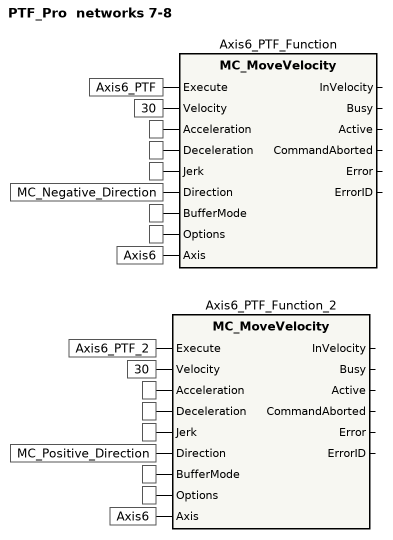
[picture p48: PTF_Pro (FBD) networks 7-8]
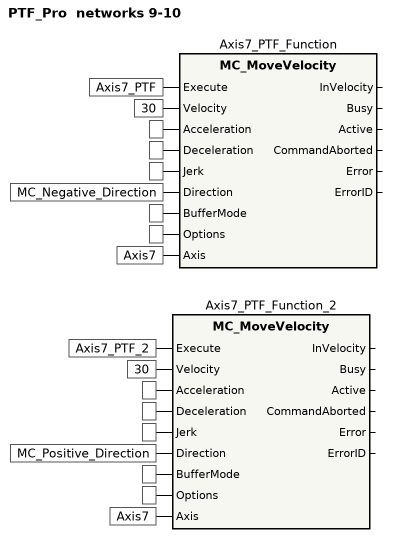
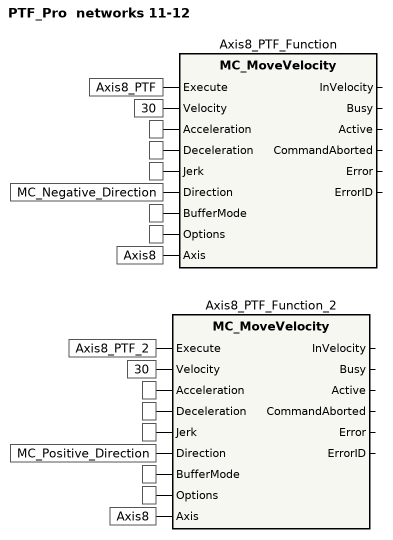
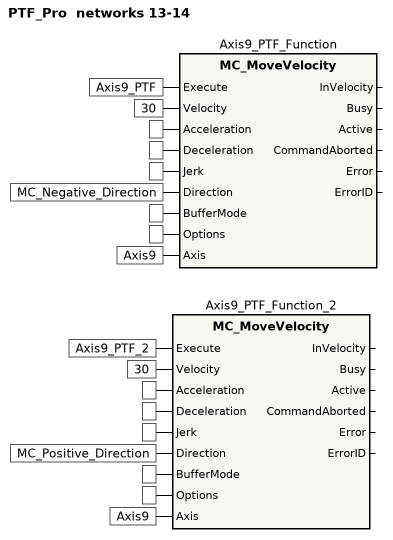
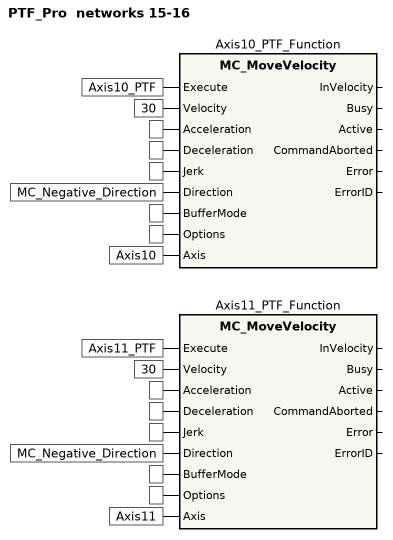
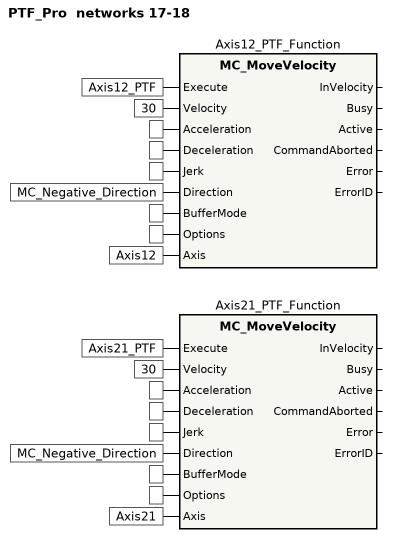
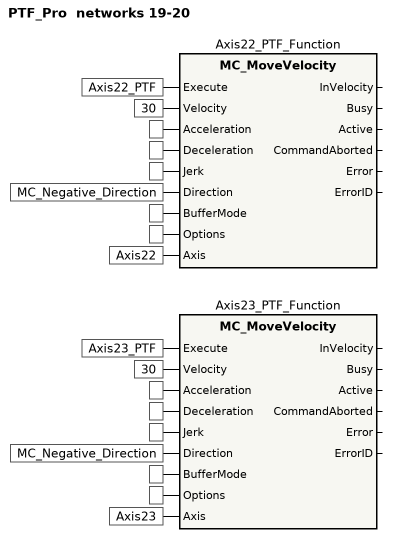
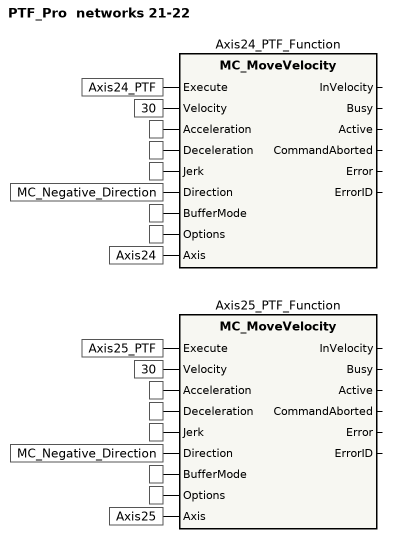
_FBD_ (* Function Block Diagram *)
NETWORK 1
	Axis1_PTF_Function:MC_MoveVelocity(Execute: Axis1_PTF, Velocity: 30, Acceleration: , Deceleration: , Jerk: , Direction: MC_Negative_Direction, BufferMode: , Options: , Axis: Axis1)
NETWORK 2
	Axis2_PTF_Function:MC_MoveVelocity(Execute: Axis2_PTF, Velocity: 30, Acceleration: , Deceleration: , Jerk: , Direction: MC_Negative_Direction, BufferMode: , Options: , Axis: Axis2)
NETWORK 3
	Axis3_PTF_Function:MC_MoveVelocity(Execute: Axis3_PTF, Velocity: 30, Acceleration: , Deceleration: , Jerk: , Direction: MC_Negative_Direction, BufferMode: , Options: , Axis: Axis3)
NETWORK 4
	Axis3_PTF_Function_2:MC_MoveVelocity(Execute: Axis3_PTF_2, Velocity: 10, Acceleration: , Deceleration: , Jerk: , Direction: MC_Positive_Direction, BufferMode: , Options: , Axis: Axis3)
NETWORK 5
	Axis4_PTF_Function:MC_MoveVelocity(Execute: Axis4_PTF, Velocity: 30, Acceleration: , Deceleration: , Jerk: , Direction: MC_Negative_Direction, BufferMode: , Options: , Axis: Axis4)
NETWORK 6
	Axis5_PTF_Function:MC_MoveVelocity(Execute: Axis5_PTF, Velocity: 30, Acceleration: , Deceleration: , Jerk: , Direction: MC_Negative_Direction, BufferMode: , Options: , Axis: Axis5)
NETWORK 7
	Axis6_PTF_Function:MC_MoveVelocity(Execute: Axis6_PTF, Velocity: 30, Acceleration: , Deceleration: , Jerk: , Direction: MC_Negative_Direction, BufferMode: , Options: , Axis: Axis6)
NETWORK 8
	Axis6_PTF_Function_2:MC_MoveVelocity(Execute: Axis6_PTF_2, Velocity: 30, Acceleration: , Deceleration: , Jerk: , Direction: MC_Positive_Direction, BufferMode: , Options: , Axis: Axis6)
NETWORK 9
	Axis7_PTF_Function:MC_MoveVelocity(Execute: Axis7_PTF, Velocity: 30, Acceleration: , Deceleration: , Jerk: , Direction: MC_Negative_Direction, BufferMode: , Options: , Axis: Axis7)
NETWORK 10
	Axis7_PTF_Function_2:MC_MoveVelocity(Execute: Axis7_PTF_2, Velocity: 30, Acceleration: , Deceleration: , Jerk: , Direction: MC_Positive_Direction, BufferMode: , Options: , Axis: Axis7)
NETWORK 11
	Axis8_PTF_Function:MC_MoveVelocity(Execute: Axis8_PTF, Velocity: 30, Acceleration: , Deceleration: , Jerk: , Direction: MC_Negative_Direction, BufferMode: , Options: , Axis: Axis8)
NETWORK 12
	Axis8_PTF_Function_2:MC_MoveVelocity(Execute: Axis8_PTF_2, Velocity: 30, Acceleration: , Deceleration: , Jerk: , Direction: MC_Positive_Direction, BufferMode: , Options: , Axis: Axis8)
NETWORK 13
	Axis9_PTF_Function:MC_MoveVelocity(Execute: Axis9_PTF, Velocity: 30, Acceleration: , Deceleration: , Jerk: , Direction: MC_Negative_Direction, BufferMode: , Options: , Axis: Axis9)
NETWORK 14
	Axis9_PTF_Function_2:MC_MoveVelocity(Execute: Axis9_PTF_2, Velocity: 30, Acceleration: , Deceleration: , Jerk: , Direction: MC_Positive_Direction, BufferMode: , Options: , Axis: Axis9)
NETWORK 15
	Axis10_PTF_Function:MC_MoveVelocity(Execute: Axis10_PTF, Velocity: 30, Acceleration: , Deceleration: , Jerk: , Direction: MC_Negative_Direction, BufferMode: , Options: , Axis: Axis10)
NETWORK 16
	Axis11_PTF_Function:MC_MoveVelocity(Execute: Axis11_PTF, Velocity: 30, Acceleration: , Deceleration: , Jerk: , Direction: MC_Negative_Direction, BufferMode: , Options: , Axis: Axis11)
NETWORK 17
	Axis12_PTF_Function:MC_MoveVelocity(Execute: Axis12_PTF, Velocity: 30, Acceleration: , Deceleration: , Jerk: , Direction: MC_Negative_Direction, BufferMode: , Options: , Axis: Axis12)
NETWORK 18
	Axis21_PTF_Function:MC_MoveVelocity(Execute: Axis21_PTF, Velocity: 30, Acceleration: , Deceleration: , Jerk: , Direction: MC_Negative_Direction, BufferMode: , Options: , Axis: Axis21)
NETWORK 19
	Axis22_PTF_Function:MC_MoveVelocity(Execute: Axis22_PTF, Velocity: 30, Acceleration: , Deceleration: , Jerk: , Direction: MC_Negative_Direction, BufferMode: , Options: , Axis: Axis22)
NETWORK 20
	Axis23_PTF_Function:MC_MoveVelocity(Execute: Axis23_PTF, Velocity: 30, Acceleration: , Deceleration: , Jerk: , Direction: MC_Negative_Direction, BufferMode: , Options: , Axis: Axis23)
NETWORK 21
	Axis24_PTF_Function:MC_MoveVelocity(Execute: Axis24_PTF, Velocity: 30, Acceleration: , Deceleration: , Jerk: , Direction: MC_Negative_Direction, BufferMode: , Options: , Axis: Axis24)
NETWORK 22
	Axis25_PTF_Function:MC_MoveVelocity(Execute: Axis25_PTF, Velocity: 30, Acceleration: , Deceleration: , Jerk: , Direction: MC_Negative_Direction, BufferMode: , Options: , Axis: Axis25)
_END_FBD_
END_PROGRAM

(* POU Other_Folder/Motion/Axis_Status_Check, FBD *)
PROGRAM Axis_Status_Check
VAR
	R1: MC_ReadStatus;
	R2: MC_ReadStatus;
	R3: MC_ReadStatus;
	R4: MC_ReadStatus;
	R5: MC_ReadStatus;
	R6: MC_ReadStatus;
	R7: MC_ReadStatus;
	R8: MC_ReadStatus;
	R9: MC_ReadStatus;
	R10: MC_ReadStatus;
	R11: MC_ReadStatus;
	R12: MC_ReadStatus;

	R21: MC_ReadStatus;
	R22: MC_ReadStatus;
	R23: MC_ReadStatus;
	R24: MC_ReadStatus;
	R25: MC_ReadStatus;
END_VAR
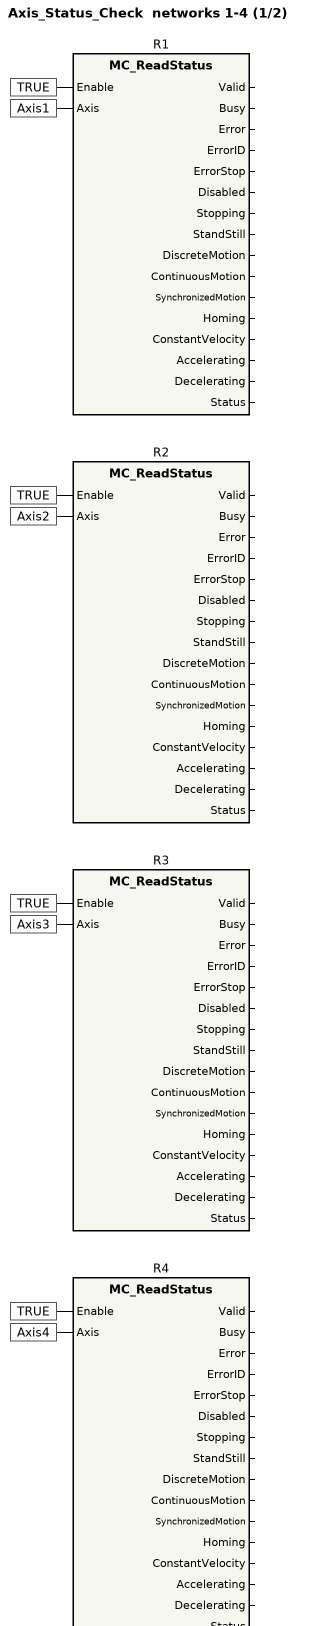
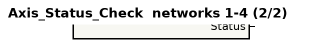
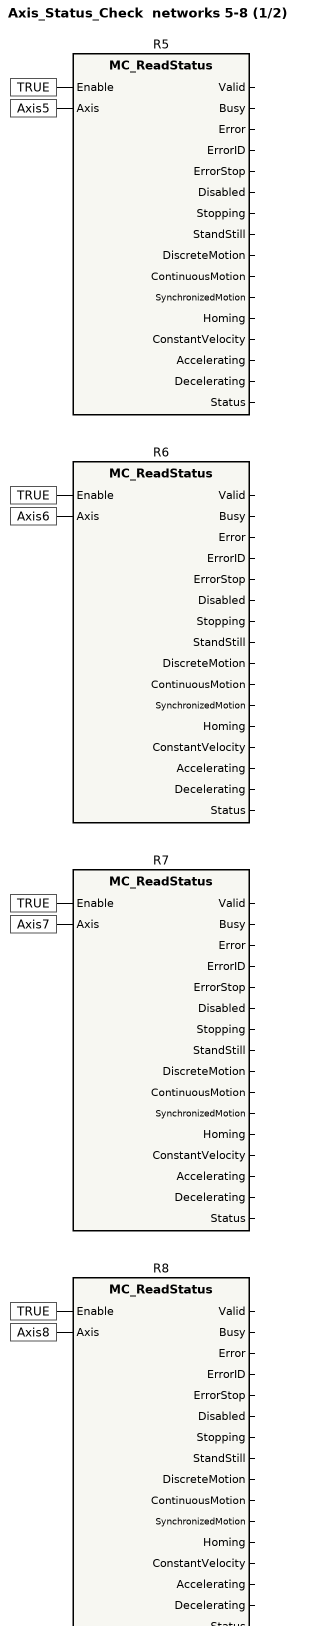
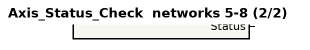
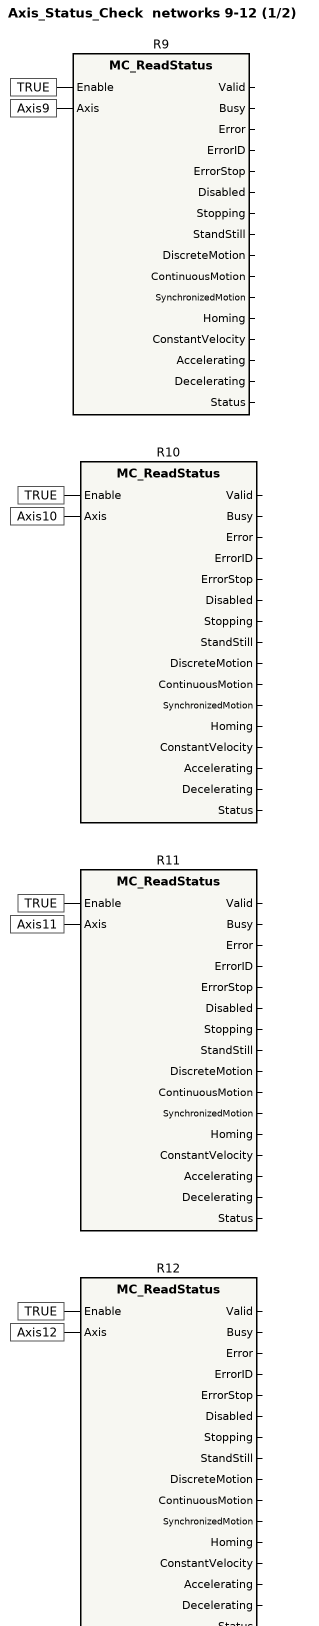
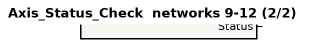
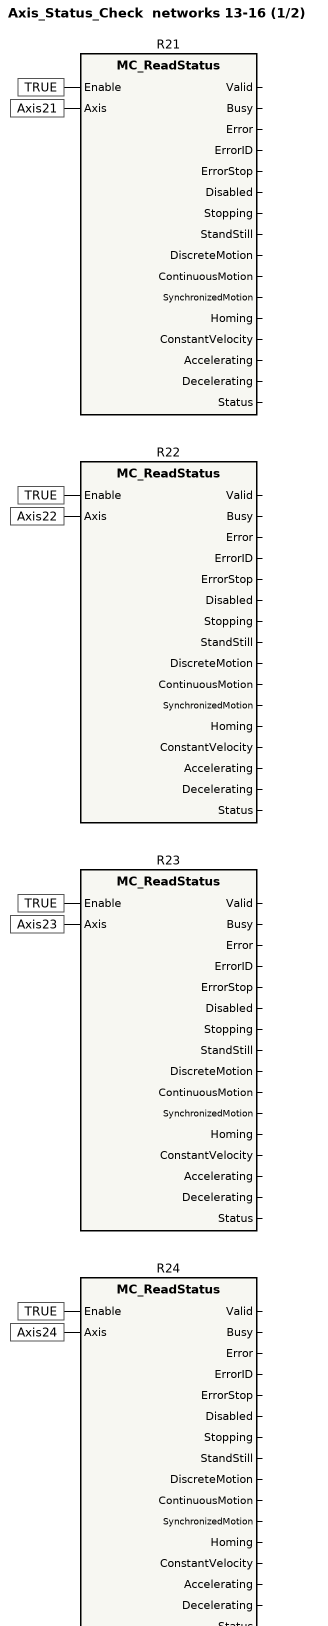
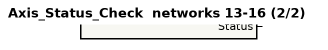
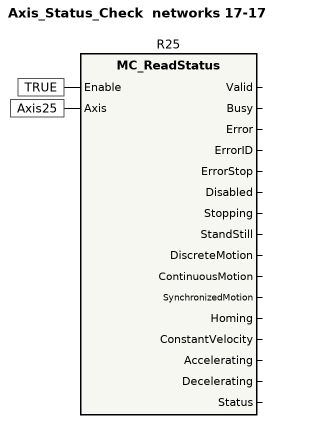
_FBD_ (* Function Block Diagram *)
NETWORK 1
	R1:MC_ReadStatus(Enable: TRUE, Axis: Axis1)
NETWORK 2
	R2:MC_ReadStatus(Enable: TRUE, Axis: Axis2)
NETWORK 3
	R3:MC_ReadStatus(Enable: TRUE, Axis: Axis3)
NETWORK 4
	R4:MC_ReadStatus(Enable: TRUE, Axis: Axis4)
NETWORK 5
	R5:MC_ReadStatus(Enable: TRUE, Axis: Axis5)
NETWORK 6
	R6:MC_ReadStatus(Enable: TRUE, Axis: Axis6)
NETWORK 7
	R7:MC_ReadStatus(Enable: TRUE, Axis: Axis7)
NETWORK 8
	R8:MC_ReadStatus(Enable: TRUE, Axis: Axis8)
NETWORK 9
	R9:MC_ReadStatus(Enable: TRUE, Axis: Axis9)
NETWORK 10
	R10:MC_ReadStatus(Enable: TRUE, Axis: Axis10)
NETWORK 11
	R11:MC_ReadStatus(Enable: TRUE, Axis: Axis11)
NETWORK 12
	R12:MC_ReadStatus(Enable: TRUE, Axis: Axis12)
NETWORK 13
	R21:MC_ReadStatus(Enable: TRUE, Axis: Axis21)
NETWORK 14
	R22:MC_ReadStatus(Enable: TRUE, Axis: Axis22)
NETWORK 15
	R23:MC_ReadStatus(Enable: TRUE, Axis: Axis23)
NETWORK 16
	R24:MC_ReadStatus(Enable: TRUE, Axis: Axis24)
NETWORK 17
	R25:MC_ReadStatus(Enable: TRUE, Axis: Axis25)
_END_FBD_
(* the same logic as Structured Text *)
(* Network 1 *)
R1(Enable := TRUE, Axis := Axis1);
(* Network 2 *)
R2(Enable := TRUE, Axis := Axis2);
(* Network 3 *)
R3(Enable := TRUE, Axis := Axis3);
(* Network 4 *)
R4(Enable := TRUE, Axis := Axis4);
(* Network 5 *)
R5(Enable := TRUE, Axis := Axis5);
(* Network 6 *)
R6(Enable := TRUE, Axis := Axis6);
(* Network 7 *)
R7(Enable := TRUE, Axis := Axis7);
(* Network 8 *)
R8(Enable := TRUE, Axis := Axis8);
(* Network 9 *)
R9(Enable := TRUE, Axis := Axis9);
(* Network 10 *)
R10(Enable := TRUE, Axis := Axis10);
(* Network 11 *)
R11(Enable := TRUE, Axis := Axis11);
(* Network 12 *)
R12(Enable := TRUE, Axis := Axis12);
(* Network 13 *)
R21(Enable := TRUE, Axis := Axis21);
(* Network 14 *)
R22(Enable := TRUE, Axis := Axis22);
(* Network 15 *)
R23(Enable := TRUE, Axis := Axis23);
(* Network 16 *)
R24(Enable := TRUE, Axis := Axis24);
(* Network 17 *)
R25(Enable := TRUE, Axis := Axis25);
END_PROGRAM

(* POU Other_Folder/Speed_AxisStatus_IO/Axis_Status, LD *)
PROGRAM Axis_Status
VAR
END_VAR
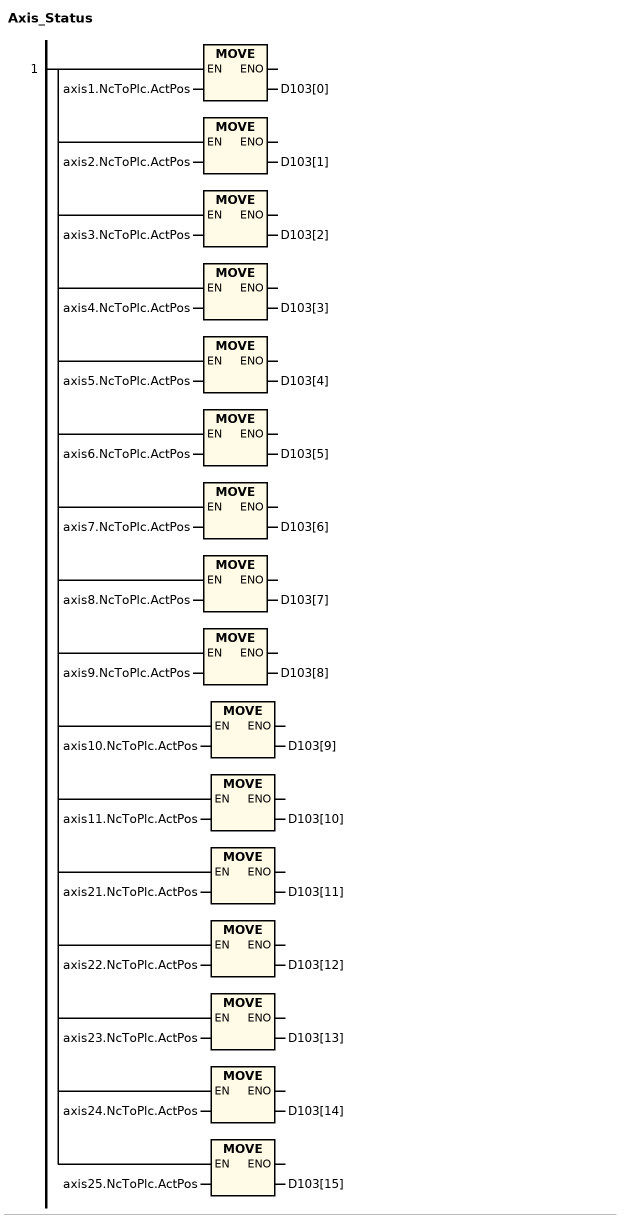
_LD_ (* Ladder Diagram *)
NETWORK 1
	*
		EN --- MOVE(axis1.NcToPlc.ActPos) => D103[0]
		EN --- MOVE(axis2.NcToPlc.ActPos) => D103[1]
		EN --- MOVE(axis3.NcToPlc.ActPos) => D103[2]
		EN --- MOVE(axis4.NcToPlc.ActPos) => D103[3]
		EN --- MOVE(axis5.NcToPlc.ActPos) => D103[4]
		EN --- MOVE(axis6.NcToPlc.ActPos) => D103[5]
		EN --- MOVE(axis7.NcToPlc.ActPos) => D103[6]
		EN --- MOVE(axis8.NcToPlc.ActPos) => D103[7]
		EN --- MOVE(axis9.NcToPlc.ActPos) => D103[8]
		EN --- MOVE(axis10.NcToPlc.ActPos) => D103[9]
		EN --- MOVE(axis11.NcToPlc.ActPos) => D103[10]
		EN --- MOVE(axis21.NcToPlc.ActPos) => D103[11]
		EN --- MOVE(axis22.NcToPlc.ActPos) => D103[12]
		EN --- MOVE(axis23.NcToPlc.ActPos) => D103[13]
		EN --- MOVE(axis24.NcToPlc.ActPos) => D103[14]
		EN --- MOVE(axis25.NcToPlc.ActPos) => D103[15]
_END_LD_
(* the same logic as Structured Text *)
(* Network 1 *)
D103[0] := axis1.NcToPlc.ActPos;
D103[1] := axis2.NcToPlc.ActPos;
D103[2] := axis3.NcToPlc.ActPos;
D103[3] := axis4.NcToPlc.ActPos;
D103[4] := axis5.NcToPlc.ActPos;
D103[5] := axis6.NcToPlc.ActPos;
D103[6] := axis7.NcToPlc.ActPos;
D103[7] := axis8.NcToPlc.ActPos;
D103[8] := axis9.NcToPlc.ActPos;
D103[9] := axis10.NcToPlc.ActPos;
D103[10] := axis11.NcToPlc.ActPos;
D103[11] := axis21.NcToPlc.ActPos;
D103[12] := axis22.NcToPlc.ActPos;
D103[13] := axis23.NcToPlc.ActPos;
D103[14] := axis24.NcToPlc.ActPos;
D103[15] := axis25.NcToPlc.ActPos;
END_PROGRAM

(* POU Other_Folder/Speed_AxisStatus_IO/Limit_Mapping, LD *)
PROGRAM Limit_Mapping
VAR

END_VAR
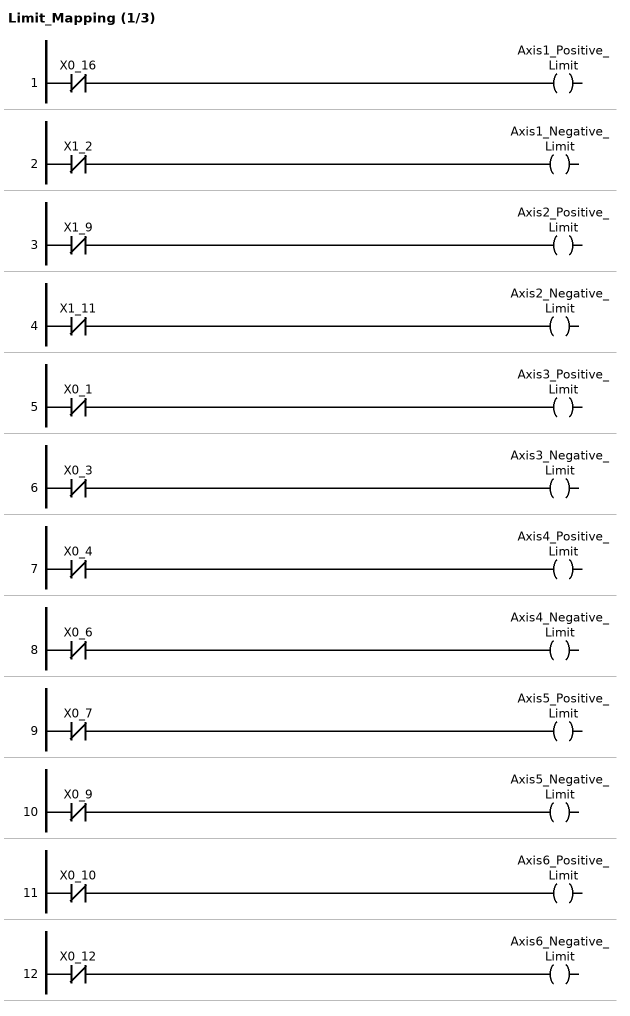
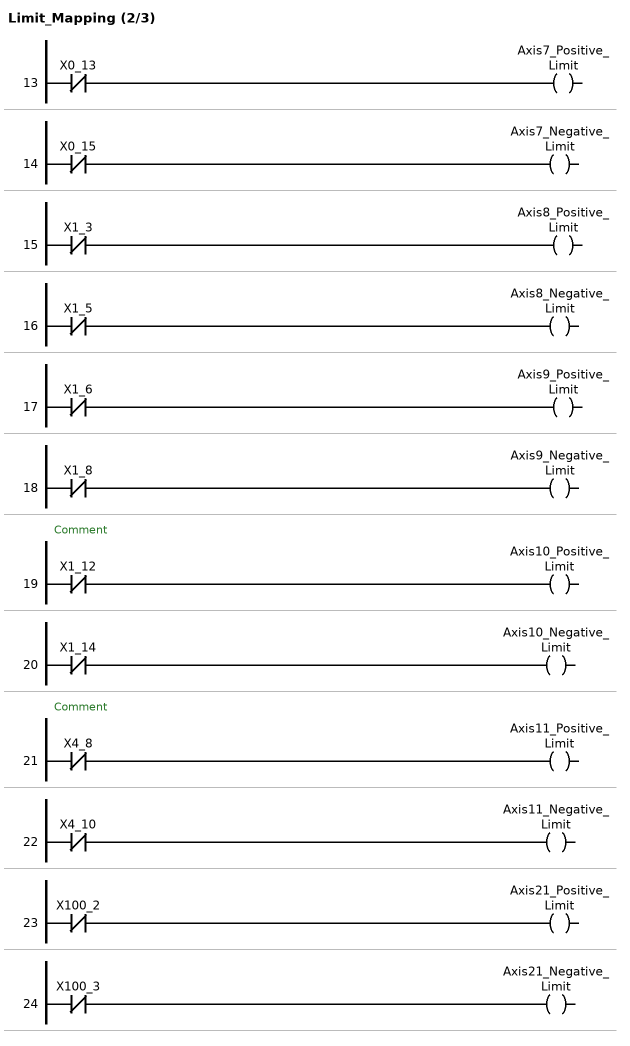
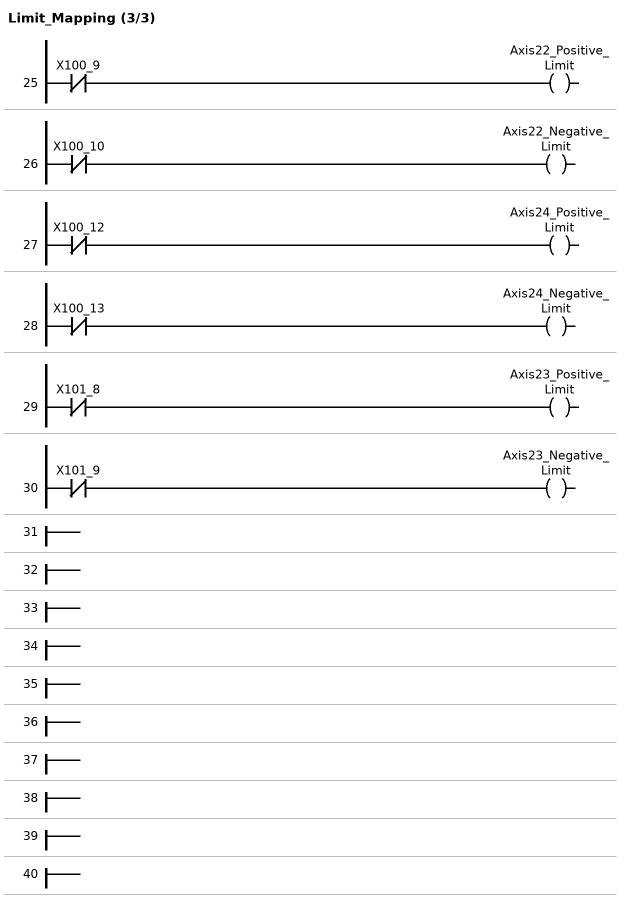
_LD_ (* Ladder Diagram *)
NETWORK 1
	[/X0_16] --- (Axis1_Positive_Limit)
NETWORK 2
	[/X1_2] --- (Axis1_Negative_Limit)
NETWORK 3
	[/X1_9] --- (Axis2_Positive_Limit)
NETWORK 4
	[/X1_11] --- (Axis2_Negative_Limit)
NETWORK 5
	[/X0_1] --- (Axis3_Positive_Limit)
NETWORK 6
	[/X0_3] --- (Axis3_Negative_Limit)
NETWORK 7
	[/X0_4] --- (Axis4_Positive_Limit)
NETWORK 8
	[/X0_6] --- (Axis4_Negative_Limit)
NETWORK 9
	[/X0_7] --- (Axis5_Positive_Limit)
NETWORK 10
	[/X0_9] --- (Axis5_Negative_Limit)
NETWORK 11
	[/X0_10] --- (Axis6_Positive_Limit)
NETWORK 12
	[/X0_12] --- (Axis6_Negative_Limit)
NETWORK 13
	[/X0_13] --- (Axis7_Positive_Limit)
NETWORK 14
	[/X0_15] --- (Axis7_Negative_Limit)
NETWORK 15
	[/X1_3] --- (Axis8_Positive_Limit)
NETWORK 16
	[/X1_5] --- (Axis8_Negative_Limit)
NETWORK 17
	[/X1_6] --- (Axis9_Positive_Limit)
NETWORK 18
	[/X1_8] --- (Axis9_Negative_Limit)
NETWORK 19 (* Comment *)
	[/X1_12] --- (Axis10_Positive_Limit)
NETWORK 20
	[/X1_14] --- (Axis10_Negative_Limit)
NETWORK 21 (* Comment *)
	[/X4_8] --- (Axis11_Positive_Limit)
NETWORK 22
	[/X4_10] --- (Axis11_Negative_Limit)
NETWORK 23
	[/X100_2] --- (Axis21_Positive_Limit)
NETWORK 24
	[/X100_3] --- (Axis21_Negative_Limit)
NETWORK 25
	[/X100_9] --- (Axis22_Positive_Limit)
NETWORK 26
	[/X100_10] --- (Axis22_Negative_Limit)
NETWORK 27
	[/X100_12] --- (Axis24_Positive_Limit)
NETWORK 28
	[/X100_13] --- (Axis24_Negative_Limit)
NETWORK 29
	[/X101_8] --- (Axis23_Positive_Limit)
NETWORK 30
	[/X101_9] --- (Axis23_Negative_Limit)
NETWORK 31
	*
NETWORK 32
	*
NETWORK 33
	*
NETWORK 34
	*
NETWORK 35
	*
NETWORK 36
	*
NETWORK 37
	*
NETWORK 38
	*
NETWORK 39
	*
NETWORK 40
	*
_END_LD_
(* the same logic as Structured Text *)
(* Network 1 *)
Axis1_Positive_Limit := NOT X0_16;
(* Network 2 *)
Axis1_Negative_Limit := NOT X1_2;
(* Network 3 *)
Axis2_Positive_Limit := NOT X1_9;
(* Network 4 *)
Axis2_Negative_Limit := NOT X1_11;
(* Network 5 *)
Axis3_Positive_Limit := NOT X0_1;
(* Network 6 *)
Axis3_Negative_Limit := NOT X0_3;
(* Network 7 *)
Axis4_Positive_Limit := NOT X0_4;
(* Network 8 *)
Axis4_Negative_Limit := NOT X0_6;
(* Network 9 *)
Axis5_Positive_Limit := NOT X0_7;
(* Network 10 *)
Axis5_Negative_Limit := NOT X0_9;
(* Network 11 *)
Axis6_Positive_Limit := NOT X0_10;
(* Network 12 *)
Axis6_Negative_Limit := NOT X0_12;
(* Network 13 *)
Axis7_Positive_Limit := NOT X0_13;
(* Network 14 *)
Axis7_Negative_Limit := NOT X0_15;
(* Network 15 *)
Axis8_Positive_Limit := NOT X1_3;
(* Network 16 *)
Axis8_Negative_Limit := NOT X1_5;
(* Network 17 *)
Axis9_Positive_Limit := NOT X1_6;
(* Network 18 *)
Axis9_Negative_Limit := NOT X1_8;
(* Network 19: Comment *)
Axis10_Positive_Limit := NOT X1_12;
(* Network 20 *)
Axis10_Negative_Limit := NOT X1_14;
(* Network 21: Comment *)
Axis11_Positive_Limit := NOT X4_8;
(* Network 22 *)
Axis11_Negative_Limit := NOT X4_10;
(* Network 23 *)
Axis21_Positive_Limit := NOT X100_2;
(* Network 24 *)
Axis21_Negative_Limit := NOT X100_3;
(* Network 25 *)
Axis22_Positive_Limit := NOT X100_9;
(* Network 26 *)
Axis22_Negative_Limit := NOT X100_10;
(* Network 27 *)
Axis24_Positive_Limit := NOT X100_12;
(* Network 28 *)
Axis24_Negative_Limit := NOT X100_13;
(* Network 29 *)
Axis23_Positive_Limit := NOT X101_8;
(* Network 30 *)
Axis23_Negative_Limit := NOT X101_9;
(* Network 31 *)
(* Network 32 *)
(* Network 33 *)
(* Network 34 *)
(* Network 35 *)
(* Network 36 *)
(* Network 37 *)
(* Network 38 *)
(* Network 39 *)
(* Network 40 *)
END_PROGRAM

(* POU Other_Folder/Speed_AxisStatus_IO/Speed_Setting, ST *)
PROGRAM Speed_Setting
VAR
	UP1: R_TRIG;
	UP2: R_TRIG;
	UP3: R_TRIG;

	step: INT;
END_VAR
CASE step OF
0:
step:=1;

1:
UP1(CLK:=M100 , Q=> );
UP2(CLK:=M101 , Q=> );
UP3(CLK:=M102 , Q=> );
(*调速选择*)
IF UP1.Q THEN(*低速*)
D11:=D100[0];D12:=D100[1];D13:=D100[2];D14:=D100[3];D15:=D100[4];
D16:=D100[5];D17:=D100[6];D18:=D100[7];D19:=D100[8];D20:=D100[9];D2_1:=D100[10];
V211:=D100[11];V221:=D100[12];V231:=D100[13];V241:=D100[14];V251:=D100[15];
step:=10;
END_IF
IF UP2.Q THEN(*中速*)
D11:=D101[0];D12:=D101[1];D13:=D101[2];D14:=D101[3];D15:=D101[4];
D16:=D101[5];D17:=D101[6];D18:=D101[7];D19:=D101[8];D20:=D101[9];D2_1:=D101[10];
V211:=D101[11];V221:=D101[12];V231:=D101[13];V241:=D101[14];V251:=D101[15];
step:=20;
END_IF
IF UP3.Q THEN(*高速*)
D11:=D102[0];D12:=D102[1];D13:=D102[2];D14:=D102[3];D15:=D102[4];
D16:=D102[5];D17:=D102[6];D18:=D102[7];D19:=D102[8];D20:=D102[9];D2_1:=D102[10];
V211:=D102[11];V221:=D102[12];V231:=D102[13];V241:=D102[14];V251:=D102[15];
step:=30;
END_IF

10:
M101:=FALSE;
M102:=FALSE;
step:=1;

20:
M100:=FALSE;
M102:=FALSE;
step:=1;

30:
M100:=FALSE;
M101:=FALSE;
step:=1;

END_CASE
END_PROGRAM

(* POU Debug_Folder/Axis1_Debug_Model, ST *)
PROGRAM Axis1_Debug_Model
VAR
	UP1: R_TRIG;
	UP2: R_TRIG;
	UP3: R_TRIG;
	UP4: R_TRIG;
	step:INT;
END_VAR
UP1(CLK:=Axis1_debug_trigger , Q=> );

CASE step OF
0:
IF UP1.Q THEN
step:=1;
END_IF;

1:
(*点动加-----------
点动减------------
手动点动-----------*)
UP2(CLK:=Axis1_mov_add , Q=> );
UP3(CLK:=Axis1_mov_sub , Q=> );
UP4(CLK:=Axis1_mov_line , Q=> );

IF UP2.Q AND Debug_Model AND Axis1_Poweron AND NOT Total_Pause THEN
D1:=Axis1.NcToPlc.ActPos+D200;
Axis1_mov_add:=FALSE;
step:=10;
ELSE
Axis1_mov_add:=FALSE;
Axis1_MoveAbsolute:=FALSE;
END_IF

IF UP3.Q AND Debug_Model AND Axis1_Poweron AND NOT Total_Pause THEN
D1:=Axis1.NcToPlc.ActPos-D200;
Axis1_mov_sub:=FALSE;
step:=10;
ELSE
Axis1_mov_sub:=FALSE;
Axis1_MoveAbsolute:=FALSE;
END_IF

IF UP4.Q AND Debug_Model AND Axis1_Poweron  AND NOT Total_Pause THEN
D1:=D201;
Axis1_mov_line:=FALSE;
step:=10;
ELSE
Axis1_mov_line:=FALSE;
Axis1_MoveAbsolute:=FALSE;
END_IF

10:
Axis1_MoveAbsolute:=TRUE;
IF Axis1_Abs_Function.Done THEN
Axis1_MoveAbsolute:=FALSE;
step:=1;
END_IF

END_CASE

IF Axis1_mov_add THEN
Axis1_mov_add:=FALSE;
END_IF
IF Axis1_mov_sub THEN
Axis1_mov_sub:=FALSE;
END_IF
IF Axis1_mov_line THEN
Axis1_mov_line:=FALSE;
END_IF


IF NOT Debug_Model  THEN
Axis1_debug_trigger:=FALSE;
step:=0;
END_IF

IF Total_Emergency THEN
Axis1_debug_trigger:=FALSE;
Axis1_mov_add:=FALSE;
Axis1_mov_sub:=FALSE;
Axis1_mov_line:=FALSE;
Axis1_MoveAbsolute:=FALSE;
step:=0;
END_IF
END_PROGRAM

(* POU Debug_Folder/Axis2_Debug_Model, ST *)
PROGRAM Axis2_Debug_Model
VAR
	UP1: R_TRIG;
	UP2: R_TRIG;
	UP3: R_TRIG;
	UP4: R_TRIG;
	step:INT;

END_VAR
UP1(CLK:=Axis2_debug_trigger , Q=> );

CASE step OF
0:
IF UP1.Q THEN
step:=1;
END_IF;

1:
UP2(CLK:=Axis2_mov_add , Q=> );
UP3(CLK:=Axis2_mov_sub , Q=> );
UP4(CLK:=Axis2_mov_line , Q=> );

IF UP2.Q AND Debug_Model AND Axis2_Poweron AND NOT Total_Pause THEN
D2:=Axis2.NcToPlc.ActPos+D200;
Axis2_mov_add:=FALSE;
step:=10;
ELSE
Axis2_mov_add:=FALSE;
Axis2_MoveAbsolute:=FALSE;
END_IF

IF UP3.Q AND Debug_Model AND Axis2_Poweron AND NOT Total_Pause THEN
D2:=Axis2.NcToPlc.ActPos-D200;
Axis2_mov_sub:=FALSE;
step:=10;
ELSE
Axis2_mov_sub:=FALSE;
Axis2_MoveAbsolute:=FALSE;
END_IF

IF UP4.Q AND Debug_Model AND Axis2_Poweron AND NOT Total_Pause THEN
D2:=D202;
Axis2_mov_line:=FALSE;
step:=10;
ELSE
Axis2_mov_line:=FALSE;
Axis2_MoveAbsolute:=FALSE;
END_IF

10:
Axis2_MoveAbsolute:=TRUE;
IF Axis2_Abs_Function.Done THEN
Axis2_MoveAbsolute:=FALSE;
step:=1;
END_IF

END_CASE

IF Axis2_mov_add THEN
Axis2_mov_add:=FALSE;
END_IF
IF Axis2_mov_sub THEN
Axis2_mov_sub:=FALSE;
END_IF
IF Axis2_mov_line THEN
Axis2_mov_line:=FALSE;
END_IF


IF NOT Debug_Model  THEN
Axis2_debug_trigger:=FALSE;
step:=0;
END_IF

IF Total_Emergency THEN
Axis2_debug_trigger:=FALSE;
Axis2_mov_add:=FALSE;
Axis2_mov_sub:=FALSE;
Axis2_mov_line:=FALSE;
Axis2_MoveAbsolute:=FALSE;
step:=0;
END_IF
END_PROGRAM

(* POU Debug_Folder/Axis3_Debug_Model, ST *)
PROGRAM Axis3_Debug_Model
VAR
	UP1: R_TRIG;
	UP2: R_TRIG;
	UP3: R_TRIG;
	UP4: R_TRIG;
	step:INT;
END_VAR
UP1(CLK:=Axis3_debug_trigger , Q=> );

CASE step OF
0:
IF UP1.Q THEN
step:=1;
END_IF;

1:
UP2(CLK:=Axis3_mov_add , Q=> );
UP3(CLK:=Axis3_mov_sub , Q=> );
UP4(CLK:=Axis3_mov_line , Q=> );

IF UP2.Q AND Debug_Model AND Axis3_Poweron AND NOT Total_Pause THEN
D3:=Axis3.NcToPlc.ActPos+D200;
Axis3_mov_add:=FALSE;
step:=10;
ELSE
Axis3_mov_add:=FALSE;
Axis3_MoveAbsolute:=FALSE;
END_IF

IF UP3.Q AND Debug_Model AND Axis3_Poweron AND NOT Total_Pause THEN
D3:=Axis3.NcToPlc.ActPos-D200;
Axis3_mov_sub:=FALSE;
step:=10;
ELSE
Axis3_mov_sub:=FALSE;
Axis3_MoveAbsolute:=FALSE;
END_IF

IF UP4.Q AND Debug_Model AND Axis3_Poweron AND NOT Total_Pause THEN
D3:=D203;
Axis3_mov_line:=FALSE;
step:=10;
ELSE
Axis3_mov_line:=FALSE;
Axis3_MoveAbsolute:=FALSE;
END_IF

10:
Axis3_MoveAbsolute:=TRUE;
IF Axis3_Abs_Function.Done THEN
Axis3_MoveAbsolute:=FALSE;
step:=1;
END_IF

END_CASE

IF Axis3_mov_add THEN
Axis3_mov_add:=FALSE;
END_IF
IF Axis3_mov_sub THEN
Axis3_mov_sub:=FALSE;
END_IF
IF Axis3_mov_line THEN
Axis3_mov_line:=FALSE;
END_IF


IF NOT Debug_Model  THEN
Axis3_debug_trigger:=FALSE;
step:=0;
END_IF

IF Total_Emergency THEN
Axis3_debug_trigger:=FALSE;
Axis3_mov_add:=FALSE;
Axis3_mov_sub:=FALSE;
Axis3_mov_line:=FALSE;
Axis3_MoveAbsolute:=FALSE;
step:=0;
END_IF
END_PROGRAM

(* POU Debug_Folder/Axis4_Debug_Model, ST *)
PROGRAM Axis4_Debug_Model
VAR
	UP1: R_TRIG;
	UP2: R_TRIG;
	UP3: R_TRIG;
	UP4: R_TRIG;
	step:INT;
	M1:BOOL;


END_VAR
UP1(CLK:=Axis4_debug_trigger , Q=> );

CASE step OF
0:
IF UP1.Q THEN
step:=1;
END_IF;

1:
UP2(CLK:=Axis4_mov_add , Q=> );
IF UP2.Q AND Debug_Model AND Axis4_Poweron  AND NOT Total_Pause THEN
D4:=Axis4.NcToPlc.ActPos+D200;
Axis4_mov_add:=FALSE;
step:=10;
ELSE
Axis4_mov_add:=FALSE;
Axis4_MoveAbsolute:=FALSE;
END_IF


UP3(CLK:=Axis4_mov_sub , Q=> );
IF UP3.Q AND Debug_Model AND Axis4_Poweron  AND NOT Total_Pause  THEN
D4:=Axis4.NcToPlc.ActPos-D200;
Axis4_mov_sub:=FALSE;
step:=10;
ELSE
Axis4_mov_sub:=FALSE;
Axis4_MoveAbsolute:=FALSE;
END_IF


UP4(CLK:=Axis4_mov_line , Q=> );
IF UP4.Q AND Debug_Model AND Axis4_Poweron  AND NOT Total_Pause  THEN
D4:=D204;
Axis4_mov_line:=FALSE;
step:=10;
ELSE
Axis4_mov_line:=FALSE;
Axis4_MoveAbsolute:=FALSE;
END_IF


10:
Axis4_MoveAbsolute:=TRUE;
IF Axis4_Abs_Function.Done THEN
Axis4_MoveAbsolute:=FALSE;
step:=1;
END_IF


END_CASE

IF Axis4_mov_add THEN
Axis4_mov_add:=FALSE;
END_IF
IF Axis4_mov_sub THEN
Axis4_mov_sub:=FALSE;
END_IF
IF Axis4_mov_line THEN
Axis4_mov_line:=FALSE;
END_IF


IF NOT Debug_Model  THEN
Axis4_debug_trigger:=FALSE;
step:=0;
END_IF

IF Total_Emergency THEN
Axis4_debug_trigger:=FALSE;
Axis4_mov_add:=FALSE;
Axis4_mov_sub:=FALSE;
Axis4_mov_line:=FALSE;
Axis4_MoveAbsolute:=FALSE;
Axis4_1_MoveAbsolute:=FALSE;
step:=0;
END_IF
END_PROGRAM

(* POU Debug_Folder/Axis5_Debug_Model, ST *)
PROGRAM Axis5_Debug_Model
VAR
	UP1: R_TRIG;
	UP2: R_TRIG;
	UP3: R_TRIG;
	UP4: R_TRIG;
	step:INT;
END_VAR
UP1(CLK:=Axis5_debug_trigger , Q=> );

CASE step OF
0:
IF UP1.Q THEN
step:=1;
END_IF;

1:
UP2(CLK:=Axis5_mov_add , Q=> );
UP3(CLK:=Axis5_mov_sub , Q=> );
UP4(CLK:=Axis5_mov_line , Q=> );

IF UP2.Q AND Debug_Model AND Axis5_Poweron  AND NOT Total_Pause THEN
D5:=Axis5.NcToPlc.ActPos+D200;
Axis5_mov_add:=FALSE;
step:=10;
ELSE
Axis5_mov_add:=FALSE;
Axis5_MoveAbsolute:=FALSE;
END_IF

IF UP3.Q AND Debug_Model AND Axis5_Poweron AND NOT Total_Pause THEN
D5:=Axis5.NcToPlc.ActPos-D200;
Axis5_mov_sub:=FALSE;
step:=10;
ELSE
Axis5_mov_sub:=FALSE;
Axis5_MoveAbsolute:=FALSE;
END_IF

IF UP4.Q AND Debug_Model AND Axis5_Poweron  AND NOT Total_Pause THEN
D5:=D205;
Axis5_mov_line:=FALSE;
step:=10;
ELSE
Axis5_mov_line:=FALSE;
Axis5_MoveAbsolute:=FALSE;
END_IF

10:
Axis5_MoveAbsolute:=TRUE;
IF Axis5_Abs_Function.Done THEN
Axis5_MoveAbsolute:=FALSE;
step:=1;
END_IF

END_CASE

IF Axis5_mov_add THEN
Axis5_mov_add:=FALSE;
END_IF
IF Axis5_mov_sub THEN
Axis5_mov_sub:=FALSE;
END_IF
IF Axis5_mov_line THEN
Axis5_mov_line:=FALSE;
END_IF


IF NOT Debug_Model  THEN
Axis5_debug_trigger:=FALSE;
step:=0;
END_IF

IF Total_Emergency THEN
Axis5_debug_trigger:=FALSE;
Axis5_mov_add:=FALSE;
Axis5_mov_sub:=FALSE;
Axis5_mov_line:=FALSE;
Axis5_MoveAbsolute:=FALSE;
Axis5_1_MoveAbsolute:=FALSE;
step:=0;
END_IF
END_PROGRAM

(* POU Debug_Folder/Axis6_Debug_Model, ST *)
PROGRAM Axis6_Debug_Model
VAR
	UP1: R_TRIG;
	UP2: R_TRIG;
	UP3: R_TRIG;
	UP4: R_TRIG;
	step:INT;
END_VAR
UP1(CLK:=Axis6_debug_trigger , Q=> );

CASE step OF
0:
IF UP1.Q THEN
step:=1;
END_IF;

1:
UP2(CLK:=Axis6_mov_add , Q=> );
UP3(CLK:=Axis6_mov_sub , Q=> );
UP4(CLK:=Axis6_mov_line , Q=> );

IF UP2.Q AND Debug_Model AND Axis6_Poweron  AND NOT Total_Pause THEN
D6:=Axis6.NcToPlc.ActPos+D200;
Axis6_mov_add:=FALSE;
step:=10;
ELSE
Axis6_mov_add:=FALSE;
Axis6_MoveAbsolute:=FALSE;
END_IF

IF UP3.Q AND Debug_Model AND Axis6_Poweron AND NOT Total_Pause THEN
D6:=Axis6.NcToPlc.ActPos-D200;
Axis6_mov_sub:=FALSE;
step:=10;
ELSE
Axis6_mov_sub:=FALSE;
Axis6_MoveAbsolute:=FALSE;
END_IF

IF UP4.Q AND Debug_Model AND Axis6_Poweron  AND NOT Total_Pause THEN
D6:=D206;
Axis6_mov_line:=FALSE;
step:=10;
ELSE
Axis6_mov_line:=FALSE;
Axis6_MoveAbsolute:=FALSE;
END_IF

10:
Axis6_MoveAbsolute:=TRUE;
IF Axis6_Abs_Function.Done THEN
Axis6_MoveAbsolute:=FALSE;
step:=1;
END_IF
END_CASE

IF Axis6_mov_add THEN
Axis6_mov_add:=FALSE;
END_IF
IF Axis6_mov_sub THEN
Axis6_mov_sub:=FALSE;
END_IF
IF Axis6_mov_line THEN
Axis6_mov_line:=FALSE;
END_IF


IF NOT Debug_Model  THEN
Axis6_debug_trigger:=FALSE;
step:=0;
END_IF

IF Total_Emergency THEN
Axis6_debug_trigger:=FALSE;
Axis6_mov_add:=FALSE;
Axis6_mov_sub:=FALSE;
Axis6_mov_line:=FALSE;
Axis6_MoveAbsolute:=FALSE;
step:=0;
END_IF
END_PROGRAM

(* POU Debug_Folder/Axis7_Debug_Model, ST *)
PROGRAM Axis7_Debug_Model
VAR
	UP1: R_TRIG;
	UP2: R_TRIG;
	UP3: R_TRIG;
	UP4: R_TRIG;
	step:INT;
END_VAR
UP1(CLK:=Axis7_debug_trigger , Q=> );

CASE step OF
0:
IF UP1.Q THEN
step:=1;
END_IF;

1:
UP2(CLK:=Axis7_mov_add , Q=> );
UP3(CLK:=Axis7_mov_sub , Q=> );
UP4(CLK:=Axis7_mov_line , Q=> );

IF UP2.Q AND Debug_Model AND Axis7_Poweron  AND NOT Total_Pause THEN
D7:=Axis7.NcToPlc.ActPos+D200;
Axis7_mov_add:=FALSE;
step:=10;
ELSE
Axis7_mov_add:=FALSE;
Axis7_MoveAbsolute:=FALSE;
END_IF

IF UP3.Q AND Debug_Model AND Axis7_Poweron AND NOT Total_Pause THEN
D7:=Axis7.NcToPlc.ActPos-D200;
Axis7_mov_sub:=FALSE;
step:=10;
ELSE
Axis7_mov_sub:=FALSE;
Axis7_MoveAbsolute:=FALSE;
END_IF

IF UP4.Q AND Debug_Model AND Axis7_Poweron  AND NOT Total_Pause THEN
D7:=D207;
Axis7_mov_line:=FALSE;
step:=10;
ELSE
Axis7_mov_line:=FALSE;
Axis7_MoveAbsolute:=FALSE;
END_IF

10:
Axis7_MoveAbsolute:=TRUE;
IF Axis7_Abs_Function.Done THEN
Axis7_MoveAbsolute:=FALSE;
step:=1;
END_IF
END_CASE

IF Axis7_mov_add THEN
Axis7_mov_add:=FALSE;
END_IF
IF Axis7_mov_sub THEN
Axis7_mov_sub:=FALSE;
END_IF
IF Axis7_mov_line THEN
Axis7_mov_line:=FALSE;
END_IF


IF NOT Debug_Model  THEN
Axis7_debug_trigger:=FALSE;
step:=0;
END_IF

IF Total_Emergency THEN
Axis7_debug_trigger:=FALSE;
Axis7_mov_add:=FALSE;
Axis7_mov_sub:=FALSE;
Axis7_mov_line:=FALSE;
Axis7_MoveAbsolute:=FALSE;
step:=0;
END_IF
END_PROGRAM

(* POU Debug_Folder/Axis8_Debug_Model, ST *)
PROGRAM Axis8_Debug_Model
VAR
	UP1: R_TRIG;
	UP2: R_TRIG;
	UP3: R_TRIG;
	UP4: R_TRIG;
	step:INT;
END_VAR
UP1(CLK:=Axis8_debug_trigger , Q=> );

CASE step OF
0:
IF UP1.Q THEN
step:=1;
END_IF;

1:
UP2(CLK:=Axis8_mov_add , Q=> );
UP3(CLK:=Axis8_mov_sub , Q=> );
UP4(CLK:=Axis8_mov_line , Q=> );

IF UP2.Q AND Debug_Model AND Axis8_Poweron  AND NOT Total_Pause THEN
D8:=Axis8.NcToPlc.ActPos+D200;
Axis8_mov_add:=FALSE;
step:=10;
ELSE
Axis8_mov_add:=FALSE;
Axis8_MoveAbsolute:=FALSE;
END_IF

IF UP3.Q AND Debug_Model AND Axis8_Poweron AND NOT Total_Pause THEN
D8:=Axis8.NcToPlc.ActPos-D200;
Axis8_mov_sub:=FALSE;
step:=10;
ELSE
Axis8_mov_sub:=FALSE;
Axis8_MoveAbsolute:=FALSE;
END_IF

IF UP4.Q AND Debug_Model AND Axis8_Poweron  AND NOT Total_Pause THEN
D8:=D208;
Axis8_mov_line:=FALSE;
step:=10;
ELSE
Axis8_mov_line:=FALSE;
Axis8_MoveAbsolute:=FALSE;
END_IF

10:
Axis8_MoveAbsolute:=TRUE;
IF Axis8_Abs_Function.Done THEN
Axis8_MoveAbsolute:=FALSE;
step:=1;
END_IF
END_CASE

IF Axis8_mov_add THEN
Axis8_mov_add:=FALSE;
END_IF
IF Axis8_mov_sub THEN
Axis8_mov_sub:=FALSE;
END_IF
IF Axis8_mov_line THEN
Axis8_mov_line:=FALSE;
END_IF


IF NOT Debug_Model  THEN
Axis8_debug_trigger:=FALSE;
step:=0;
END_IF

IF Total_Emergency THEN
Axis8_debug_trigger:=FALSE;
Axis8_mov_add:=FALSE;
Axis8_mov_sub:=FALSE;
Axis8_mov_line:=FALSE;
Axis8_MoveAbsolute:=FALSE;
step:=0;
END_IF
END_PROGRAM

(* POU Debug_Folder/Axis9_Debug_Model, ST *)
PROGRAM Axis9_Debug_Model
VAR
	UP1: R_TRIG;
	UP2: R_TRIG;
	UP3: R_TRIG;
	UP4: R_TRIG;
	step:INT;
END_VAR
UP1(CLK:=Axis9_debug_trigger , Q=> );

CASE step OF
0:
IF UP1.Q THEN
step:=1;
END_IF;

1:
UP2(CLK:=Axis9_mov_add , Q=> );
UP3(CLK:=Axis9_mov_sub , Q=> );
UP4(CLK:=Axis9_mov_line , Q=> );

IF UP2.Q AND Debug_Model AND Axis9_Poweron  AND NOT Total_Pause THEN
D9:=Axis9.NcToPlc.ActPos+D200;
Axis9_mov_add:=FALSE;
step:=10;
ELSE
Axis9_mov_add:=FALSE;
Axis9_MoveAbsolute:=FALSE;
END_IF

IF UP3.Q AND Debug_Model AND Axis9_Poweron AND NOT Total_Pause THEN
D9:=Axis9.NcToPlc.ActPos-D200;
Axis9_mov_sub:=FALSE;
step:=10;
ELSE
Axis9_mov_sub:=FALSE;
Axis9_MoveAbsolute:=FALSE;
END_IF

IF UP4.Q AND Debug_Model AND Axis9_Poweron  AND NOT Total_Pause THEN
D9:=D209;
Axis9_mov_line:=FALSE;
step:=10;
ELSE
Axis9_mov_line:=FALSE;
Axis9_MoveAbsolute:=FALSE;
END_IF

10:
Axis9_MoveAbsolute:=TRUE;
IF Axis9_Abs_Function.Done THEN
Axis9_MoveAbsolute:=FALSE;
step:=1;
END_IF
END_CASE

IF Axis9_mov_add THEN
Axis9_mov_add:=FALSE;
END_IF
IF Axis9_mov_sub THEN
Axis9_mov_sub:=FALSE;
END_IF
IF Axis9_mov_line THEN
Axis9_mov_line:=FALSE;
END_IF


IF NOT Debug_Model  THEN
Axis9_debug_trigger:=FALSE;
step:=0;
END_IF

IF Total_Emergency THEN
Axis9_debug_trigger:=FALSE;
Axis9_mov_add:=FALSE;
Axis9_mov_sub:=FALSE;
Axis9_mov_line:=FALSE;
Axis9_MoveAbsolute:=FALSE;
step:=0;
END_IF
END_PROGRAM

(* POU Debug_Folder/Axis10_Debug_Model, ST *)
PROGRAM Axis10_Debug_Model
VAR
	UP1: R_TRIG;
	UP2: R_TRIG;
	UP3: R_TRIG;
	UP4: R_TRIG;
	step:INT;
END_VAR
UP1(CLK:=Axis10_debug_trigger , Q=> );

CASE step OF
0:
IF UP1.Q THEN
step:=1;
END_IF;

1:
UP2(CLK:=Axis10_mov_add , Q=> );
UP3(CLK:=Axis10_mov_sub , Q=> );
UP4(CLK:=Axis10_mov_line , Q=> );

IF UP2.Q AND Debug_Model AND Axis10_Poweron  AND NOT Total_Pause THEN
D10:=Axis10.NcToPlc.ActPos+D200;
Axis10_mov_add:=FALSE;
step:=10;
ELSE
Axis10_mov_add:=FALSE;
Axis10_MoveAbsolute:=FALSE;
END_IF

IF UP3.Q AND Debug_Model AND Axis10_Poweron AND NOT Total_Pause THEN
D10:=Axis10.NcToPlc.ActPos-D200;
Axis10_mov_sub:=FALSE;
step:=10;
ELSE
Axis10_mov_sub:=FALSE;
Axis10_MoveAbsolute:=FALSE;
END_IF

IF UP4.Q AND Debug_Model AND Axis10_Poweron  AND NOT Total_Pause THEN
D10:=D210;
Axis10_mov_line:=FALSE;
step:=10;
ELSE
Axis10_mov_line:=FALSE;
Axis10_MoveAbsolute:=FALSE;
END_IF

10:
Axis10_MoveAbsolute:=TRUE;
IF Axis10_Abs_Function.Done THEN
Axis10_MoveAbsolute:=FALSE;
step:=1;
END_IF
END_CASE

IF Axis10_mov_add THEN
Axis10_mov_add:=FALSE;
END_IF
IF Axis10_mov_sub THEN
Axis10_mov_sub:=FALSE;
END_IF
IF Axis10_mov_line THEN
Axis10_mov_line:=FALSE;
END_IF


IF NOT Debug_Model  THEN
Axis10_debug_trigger:=FALSE;
step:=0;
END_IF

IF Total_Emergency THEN
Axis10_debug_trigger:=FALSE;
Axis10_mov_add:=FALSE;
Axis10_mov_sub:=FALSE;
Axis10_mov_line:=FALSE;
Axis10_MoveAbsolute:=FALSE;
step:=0;
END_IF
END_PROGRAM

(* POU Debug_Folder/Axis11_Debug_Model, ST *)
PROGRAM Axis11_Debug_Model
VAR

	UP1: R_TRIG;
	UP2: R_TRIG;
	UP3: R_TRIG;
	UP4: R_TRIG;
	step:INT;
END_VAR
UP1(CLK:=Axis11_debug_trigger , Q=> );

CASE step OF
0:
IF UP1.Q THEN
step:=1;
END_IF;

1:
UP2(CLK:=Axis11_mov_add , Q=> );
UP3(CLK:=Axis11_mov_sub , Q=> );
UP4(CLK:=Axis11_mov_line , Q=> );

IF UP2.Q AND Debug_Model AND Axis11_Poweron  AND NOT Total_Pause THEN
D1_1:=Axis11.NcToPlc.ActPos+D200;
Axis11_mov_add:=FALSE;
step:=10;
ELSE
Axis11_mov_add:=FALSE;
Axis11_MoveAbsolute:=FALSE;
END_IF

IF UP3.Q AND Debug_Model AND Axis11_Poweron AND NOT Total_Pause THEN
D1_1:=Axis11.NcToPlc.ActPos-D200;
Axis11_mov_sub:=FALSE;
step:=10;
ELSE
Axis11_mov_sub:=FALSE;
Axis11_MoveAbsolute:=FALSE;
END_IF

IF UP4.Q AND Debug_Model AND Axis11_Poweron  AND NOT Total_Pause THEN
D1_1:=D211;
Axis11_mov_line:=FALSE;
step:=10;
ELSE
Axis11_mov_line:=FALSE;
Axis11_MoveAbsolute:=FALSE;
END_IF

10:
Axis11_MoveAbsolute:=TRUE;
IF Axis11_Abs_Function.Done THEN
Axis11_MoveAbsolute:=FALSE;
step:=1;
END_IF
END_CASE

IF Axis11_mov_add THEN
Axis11_mov_add:=FALSE;
END_IF
IF Axis11_mov_sub THEN
Axis11_mov_sub:=FALSE;
END_IF
IF Axis11_mov_line THEN
Axis11_mov_line:=FALSE;
END_IF


IF NOT Debug_Model  THEN
Axis11_debug_trigger:=FALSE;
step:=0;
END_IF

IF Total_Emergency THEN
Axis11_debug_trigger:=FALSE;
Axis11_mov_add:=FALSE;
Axis11_mov_sub:=FALSE;
Axis11_mov_line:=FALSE;
Axis11_MoveAbsolute:=FALSE;
step:=0;
END_IF
END_PROGRAM

(* POU Debug_Folder/Others_Debug_Model, LD *)
PROGRAM Others_Debug_Model
VAR
END_VAR
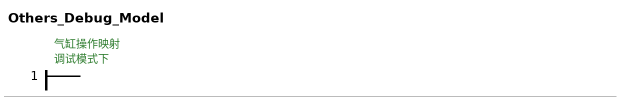
_LD_ (* Ladder Diagram *)
NETWORK 1 (* 气缸操作映射 / 调试模式下 *)
	*
_END_LD_
(* the same logic as Structured Text *)
(* Network 1: 气缸操作映射 / 调试模式下 *)
END_PROGRAM

(* POU Other_Folder/Akam_Stop_Message/Initialization_Folder/Debug12, LD *)
	PROGRAM Debug12
VAR
	t1: TON;
END_VAR
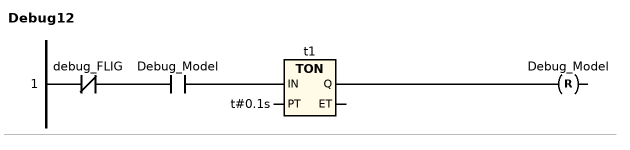
_LD_ (* Ladder Diagram *)
NETWORK 1
	[/debug_FLIG] - [Debug_Model] - t1:TON(IN: *, PT: t#0.1s) --- (R Debug_Model)
_END_LD_
(* the same logic as Structured Text *)
(* Network 1 *)
t1(IN := NOT debug_FLIG AND Debug_Model, PT := t#0.1s);
IF t1.Q THEN Debug_Model := FALSE; END_IF;
END_PROGRAM

(* POU Run_Main_Folder/Feed_alam_status, LD *)
PROGRAM Feed_alam_status
VAR


END_VAR
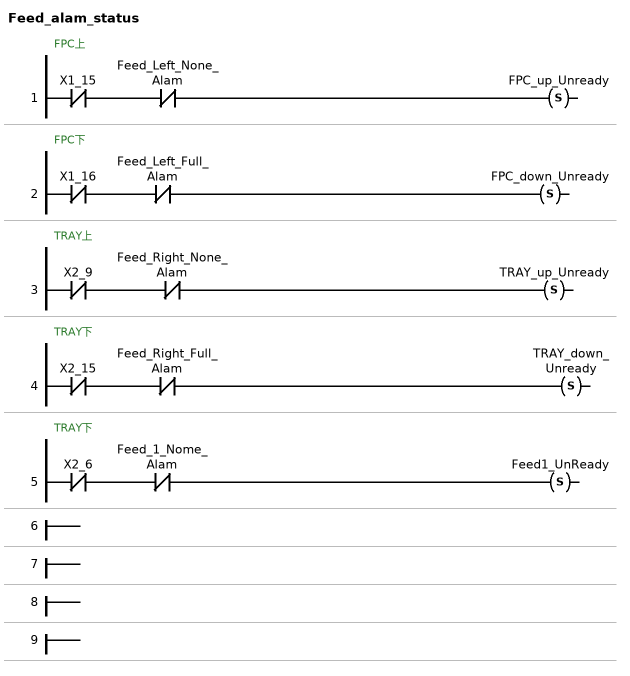
_LD_ (* Ladder Diagram *)
NETWORK 1 (* FPC上 *)
	[/X1_15] - [/Feed_Left_None_Alam] --- (S FPC_up_Unready)
NETWORK 2 (* FPC下 *)
	[/X1_16] - [/Feed_Left_Full_Alam] --- (S FPC_down_Unready)
NETWORK 3 (* TRAY上 *)
	[/X2_9] - [/Feed_Right_None_Alam] --- (S TRAY_up_Unready)
NETWORK 4 (* TRAY下 *)
	[/X2_15] - [/Feed_Right_Full_Alam] --- (S TRAY_down_Unready)
NETWORK 5 (* TRAY下 *)
	[/X2_6] - [/Feed_1_Nome_Alam] --- (S Feed1_UnReady)
NETWORK 6
	*
NETWORK 7
	*
NETWORK 8
	*
NETWORK 9
	*
_END_LD_
(* the same logic as Structured Text *)
(* Network 1: FPC上 *)
IF NOT X1_15 AND NOT Feed_Left_None_Alam THEN FPC_up_Unready := TRUE; END_IF;
(* Network 2: FPC下 *)
IF NOT X1_16 AND NOT Feed_Left_Full_Alam THEN FPC_down_Unready := TRUE; END_IF;
(* Network 3: TRAY上 *)
IF NOT X2_9 AND NOT Feed_Right_None_Alam THEN TRAY_up_Unready := TRUE; END_IF;
(* Network 4: TRAY下 *)
IF NOT X2_15 AND NOT Feed_Right_Full_Alam THEN TRAY_down_Unready := TRUE; END_IF;
(* Network 5: TRAY下 *)
IF NOT X2_6 AND NOT Feed_1_Nome_Alam THEN Feed1_UnReady := TRUE; END_IF;
(* Network 6 *)
(* Network 7 *)
(* Network 8 *)
(* Network 9 *)
END_PROGRAM

(* POU Other_Folder/Home_Back/Axis1_Home_Back, LD *)
PROGRAM Axis1_Home_Back
VAR
	UP1: R_TRIG;
	M1: BOOL;
	M2: BOOL;
	UP2: R_TRIG;
	T1: TON;
	M3: BOOL;
	M4: BOOL;
	DOWN1: F_TRIG;
	M20: BOOL;
END_VAR
VAR (* helpers for the ST form of the networks *)
	_p1 : BOOL;
	_p2 : BOOL;
	_p3 : BOOL;
END_VAR
